FUNCTION_BLOCK FB_ResultPrinter
VAR_INPUT
    nTestFunctionBlocksFinished : UINT;
END_VAR
VAR_OUTPUT
    bFinishedPrinting : BOOL;
END_VAR
VAR
    (* Although we can print a message no #1 prior to message no #2, the message #2 can still be displayed before
       message #1, most likely because of some delay of the ADS data. To workaround this, we add a small delay between
       transmission of the ADS messages. *)
    fbADSDelayTimer : TON := (PT := T#300MS);
    nLastPrintState : USINT := 0;
    nPrintState : USINT := 0;
END_VAR

CASE nPrintState OF
    0 :
        nLastPrintstate := nPrintState;
        nPrintState := 100;

    1 :
        Tc2_System.ADSLOGSTR(msgCtrlMask := Tc2_System.ADSLOG_MSGTYPE_ERROR,
                             msgFmtStr := '%s', strArg := '| ==========TESTS FINISHED RUNNING==========');
        nLastPrintstate := nPrintState;
        nPrintState := 100;

    2 :
        Tc2_System.ADSLOGSTR(msgCtrlMask := Tc2_System.ADSLOG_MSGTYPE_ERROR,
                             msgFmtStr := '| Total amount of test function blocks executed : %s',
                             strArg := UINT_TO_STRING(nTestFunctionBlocksFinished));
        nLastPrintstate := nPrintState;
        nPrintState := 100;

    3 :
        Tc2_System.ADSLOGSTR(msgCtrlMask := Tc2_System.ADSLOG_MSGTYPE_ERROR,
                             msgFmtStr := '| Failed asserts : %s',
                             strArg := UINT_TO_STRING(GVL_AssertResult.nAssertFailuresCount));
        nLastPrintstate := nPrintState;
        nPrintState := 100;

    4 :
        Tc2_System.ADSLOGSTR(msgCtrlMask := Tc2_System.ADSLOG_MSGTYPE_ERROR,
                             msgFmtStr := '| Successful asserts : %s',
                             strArg := UINT_TO_STRING(GVL_AssertResult.nAssertSuccessCount));
        nLastPrintstate := nPrintState;
        nPrintState := 100;

    5 :
        Tc2_System.ADSLOGSTR(msgCtrlMask := Tc2_System.ADSLOG_MSGTYPE_ERROR,
                             msgFmtStr := '%s', strArg := '| ======================================');
        nLastPrintstate := nPrintState;
        nPrintState := 100;

    6 :
        bFinishedPrinting := TRUE;

    100 :
        fbADSDelayTimer(IN := TRUE);
        IF fbADSDelayTimer.Q THEN
            fbADSDelayTimer(IN := FALSE);
            nPrintState := nLastPrintState + 1;
		END_IF

END_CASE

END_FUNCTION_BLOCK

(* stored: Version 1.1.0.1, ProductVersion 3.1.4022.12
   POU FB_ResultPrinter: Id {d14d6247-3ce3-459f-be22-6ee3520279ed}, SpecialFunc None *)
